// TwinCAT 3 PLC project PLC_Interpolation
// ProgramVersion: 3.1.4020.10
// libraries:
//   Tc2_MC2, * (Beckhoff Automation GmbH)
//   Tc2_NCI, * (Beckhoff Automation GmbH)
//   Tc2_PlcInterpolation, * (Beckhoff Automation GmbH)
//   Tc2_Standard, * (Beckhoff Automation GmbH)
//   Tc2_System, * (Beckhoff Automation GmbH)
//   Tc3_Interfaces, * (Beckhoff Automation GmbH)
//   Tc3_Module, * (Beckhoff Automation GmbH)
// project tree:
//   / Interpolation_FunctionResult.TcDUT, MAIN.TcPOU, NCIChannel.TcPOU, NCITable.TcPOU, NCI_REF.TcDUT, PlcTask.TcTTO
// (motion and I/O tree: see PLC project motion_library)
// real-time tasks:
//   TASK PlcTask: cycle T#10ms, priority 20, ADS port 350

CONFIGURATION PLC_Interpolation
    RESOURCE PLC ON TwinCAT3
        TASK PlcTask(INTERVAL := T#10ms, PRIORITY := 20);
        PROGRAM MAIN WITH PlcTask : MAIN;
    END_RESOURCE
END_CONFIGURATION

// ---- Interpolation_FunctionResult.TcDUT
TYPE Interpolation_FunctionResult :
(
	ERROR := -1,
	BUSY := 0,
	DONE,
	ABORTED
);
END_TYPE

// ---- NCI_REF.TcDUT
TYPE NCI_REF :
STRUCT
	NCTOPLC_nciref AT %I* : NCTOPLC_NCICHANNEL_REF;
	PLCTONC_nciref AT %Q* : PLCTONC_NCICHANNEL_REF;
END_STRUCT
END_TYPE

// ---- MAIN.TcPOU
PROGRAM MAIN
VAR
	NCI : NCICHannel;
END_VAR

END_PROGRAM

// ---- NCIChannel.TcPOU
FUNCTION_BLOCK NCIChannel
VAR_INPUT
END_VAR
VAR_OUTPUT
END_VAR
VAR
	nciGroup	: NCI_REF;
	xyzAxis		: ARRAY[0..2] OF POINTER TO AXIS_REF;
	auxAxis		: ARRAY[0..4] OF POINTER TO AXIS_REF;
	nciInit		: CfgBuildExt3DGroup;
	stTable		: NCITable;
END_VAR

METHOD FB_init : BOOL
VAR_INPUT
	bInitRetains	: BOOL; // if TRUE, the retain variables are initialized (warm start / cold start)
	bInCopyCode		: BOOL;  // if TRUE, the instance afterwards gets moved into the copy code (online change)

	X_Axis			: POINTER TO AXIS_REF;
	Y_Axis			: POINTER TO AXIS_REF;
	Z_Axis			: POINTER TO AXIS_REF;
	Q1_Axis			: POINTER TO AXIS_REF;
	Q2_Axis			: POINTER TO AXIS_REF;
	Q3_Axis			: POINTER TO AXIS_REF;
	Q4_Axis			: POINTER TO AXIS_REF;
	Q5_Axis			: POINTER TO AXIS_REF;
END_VAR
xyzAxis[0] := X_Axis;
xyzAxis[1] := Y_Axis;
xyzAxis[2] := Z_Axis;

auxAxis[0] := Q1_Axis;
auxAxis[1] := Q2_Axis;
auxAxis[2] := Q3_Axis;
auxAxis[3] := Q4_Axis;
auxAxis[4] := Q5_Axis;
END_METHOD

METHOD PUBLIC Initialise : Interpolation_FunctionResult
VAR_INPUT
END_VAR
nciInit(
	bExecute:= TRUE, 
	nGroupId:= NCIGroup.NCTOPLC_nciref.GrpId, 
	nXAxisId:= xyzAxis[0]^.NcToPlc.AxisId, 
	nYAxisId:= xyzAxis[1]^.NcToPlc.AxisId, 
	nZAxisId:= xyzAxis[2]^.NcToPlc.AxisId, 
	
	nQ1AxisId:= auxAxis[0]^.NcToPlc.AxisId, 
	nQ2AxisId:= auxAxis[1]^.NcToPlc.AxisId, 
	nQ3AxisId:= auxAxis[2]^.NcToPlc.AxisId, 
	nQ4AxisId:= auxAxis[3]^.NcToPlc.AxisId, 
	nQ5AxisId:= auxAxis[4]^.NcToPlc.AxisId, 
	tTimeOut:= T#1S
	);
	
IF NOT nciInit.bBusy AND NOT nciInit.bErr THEN
	nciInit( bExecute := FALSE );
	Initialise := Interpolation_FunctionResult.DONE;
ELSIF nciInit.bErr THEN
	Initialise := Interpolation_FunctionResult.ERROR;
ELSE
	Initialise := Interpolation_FunctionResult.BUSY;
END_IF
END_METHOD

END_FUNCTION_BLOCK

// ---- NCITable.TcPOU
FUNCTION_BLOCK NCITable
VAR_INPUT
END_VAR
VAR_OUTPUT
END_VAR
VAR
	nciTable : ST_NciFeedGroupTable;
END_VAR

;

END_FUNCTION_BLOCK
